(* PLC project Generated.project, CODESYS CODESYS V3.5 SP19 Patch 1 *)
(* stored: creationDateTime 2026-09-06T13:00:42.384826, modificationDateTime 2026-09-06T13:00:42.384826 *)

(* ======================================================================= 🧩 ST_Fault — Brique socle défaut (2 vues : live + latchée) ─────────────────────────────────────────────────────────────── 🎯 Rôle : porter l'état défaut d'un composant, applicable dans TOUS les cas (acquittable ou non), sans brique warning séparée. • Vue LIVE (Error / ErrorId) : suit la cause, retombe seule à 0. • Vue LATCHÉE (Latched / LatchedId): mémorisée au défaut, reste jusqu'au front Reset. Le choix acquittable / non-acquittable se fait PAR CAUSE (ST_FaultCause.Latching), jamais par bloc. 🔒 Sécurité : interlock TOUJOURS sur la cause brute (Error / ErrorId), jamais sur l'acquittement. Reset TOUJOURS effectif, jamais conditionné (std §9). 🧬 Composition : brique de base réutilisable — sortie de FB, struct métier, GVL. Texte IHM NON stocké ici : dérivé côté IHM depuis LatchedId / ErrorId. 📄 Doc : DOC/STDS/CODE_QUALITY_STANDARDS.md §2quinquies / §9 ======================================================================= *)
TYPE ST_Fault : STRUCT
  Error : BOOL;  (* <-- [DIAG] vue LIVE : au moins une cause présente maintenant *)
  ErrorId : WORD;  (* <-- [DIAG] bitfield des causes présentes maintenant (0 si aucune) *)
  Latched : BOOL;  (* <-- [DIAG] vue LATCHÉE : défaut non acquitté, reste jusqu'au front Reset *)
  LatchedId : WORD;  (* <-- [DIAG] ErrorId figé à l'apparition du défaut, effacé au Reset *)
END_STRUCT;
END_TYPE

(* ======================================================================= 🧩 ST_FaultCause — Cause élémentaire alimentant ST_Fault (socle FB_FaultCore) ─────────────────────────────────────────────────────────────── 🎯 Rôle : une cause exprimée EN CLAIR (BOOL + libellé), sans bitfield ni masque. Le FB métier remplit une liste (ARRAY[0..15] OF ST_FaultCause) ; le socle FB_FaultCore en déduit ST_Fault (vue live + vue latchée). 🔒 Sécurité : interlock TOUJOURS sur Active (cause brute), jamais sur le latch. Latching = TRUE → la cause ARME la vue latchée (défaut à acquitter). Latching = FALSE → la cause n'alimente que la vue live (retombe seule). Fail-safe : une cause laissée à Latching=FALSE reste visible en live — pour la rendre acquittable, il faut le déclarer explicitement. 📄 Doc : DOC/STDS/CODE_QUALITY_STANDARDS.md §2quinquies / §9 ======================================================================= *)
TYPE ST_FaultCause : STRUCT
  Active : BOOL;  (* 1 = cause présente maintenant (interlock sur cette valeur) *)
  Latching : BOOL;  (* 1 = cause à acquitter (arme Latched) ; 0 = live seulement *)
  Texte : STRING;  (* libellé prêt IHM (non stocké dans ST_Fault, dérivé côté IHM) *)
END_STRUCT;
END_TYPE

(* ======================================================================= 🛡️ FB_Encoder_Safety — Bornage physique & surveillance cohérence ─────────────────────────────────────────────────────────────── 🎯 Rôle : Bornage physique absolu [-99; +99]m et relais d'incohérence redémarrage 🔒 Polarité : EncoderIncoherent=TRUE en cas de hors bornes ou HomingSuspect 🛡️ Sécurité : Verrouillage de la position câble sûre 📄 Doc métier : DOC/AF/AF_Partie-09_Fonction_Encoder_v2.4.md ======================================================================= *)
FUNCTION_BLOCK FB_Encoder_Safety
  VAR_INPUT
    Enable : BOOL;  (* === COMMANDES & AUTORISATIONS === --> [CMD] Autorisation generale FB (TRUE=Autorise) *)
    Reset : BOOL;  (* --> [CMD] Acquittement defaut (front montant) *)
    CablePosM : REAL;  (* === MESURES & ALERTE HOMING === --> [HW] Position calculee (m, sortie FB_Encoder_Scale) *)
    HomingSuspect : BOOL;  (* --> [SAFE] Alerte incoherence redemarrage (FB_Encoder_Homing) *)
    PositionMinM : REAL := -99;  (* === REGLAGES & BORNES PHYSIQUES === --> [CFG] Plafond bornage physique bas (m) *)
    PositionMaxM : REAL := 99;  (* --> [CFG] Plafond bornage physique haut (m) *)
    BypassGlobal : BOOL := FALSE;  (* === TESTS & BYPASS === --> [TST] Neutralisation defaut de bornage pour mise en service *)
  END_VAR
  VAR_OUTPUT
    Ready : BOOL;  (* === ETATS IEC & SYNOPTIQUE === <-- [STAT] FB pret a fonctionner *)
    Fault : ST_Fault;  (* 🧩 Statut transverse (forme cible ST_Fault) *)
    CablePosMSafe : REAL;  (* === MESURES SURE & SECURITE === <-- [DIAG] Position cable instantanee transmise (m) *)
    EncoderIncoherent : BOOL;  (* <-- [SAFE] Incoherence ou hors bornes (TRUE = defaut) *)
  END_VAR
  VAR
    ResetEdge : R_TRIG;  (* === DETECTEURS DE FRONT === . [LOC] Detecteur front montant Reset *)
    instFault : FB_FaultCore;  (* === SOCLE DEFAUT (FB_FaultCore) === * [INST] Socle défaut transverse *)
    instCauses : ARRAY[0..15] OF ST_FaultCause;  (* . [LOC] Table des causes nommées *)
  END_VAR

            

// === IMPLEMENTATION ===

{region "§1 Causes & Socle Défaut (évalué en continu)"}
// 🔑 1. RESET FRONT
ResetEdge(CLK := Reset);

// 🔍 2. SURVEILLANCE BORNAGE & INCOHÉRENCE BOOT
instCauses[0].Active   := NOT BypassGlobal AND ((CablePosM < PositionMinM) OR (CablePosM > PositionMaxM));
instCauses[0].Latching := FALSE;
instCauses[0].Texte    := 'Depassement bornes physiques absolues cable';

instCauses[1].Active   := NOT BypassGlobal AND HomingSuspect;
instCauses[1].Latching := FALSE;
instCauses[1].Texte    := 'Incoherence position au redemarrage';

// Appel du socle de défaut
instFault(Enable := Enable, Reset := Reset, Causes := instCauses);
Fault := instFault.Fault;
{endregion}

{region "§2 Gate neutralisation"}
// 🛑 2. GATE
IF NOT Enable THEN
    Ready := FALSE;
    CablePosMSafe := CablePosM;
    EncoderIncoherent := FALSE;
    RETURN;
END_IF;

Ready := Enable AND NOT Fault.Latched;
{endregion}

{region "§3 Transmission mesure et sécurité"}
// 📏 3. TRANSMISSION DE LA MESURE & SÉCURITÉ
CablePosMSafe := CablePosM;
EncoderIncoherent := Fault.Error;
{endregion}

          
END_FUNCTION_BLOCK

(* ======================================================================= 🧩 FB_FaultCore — Socle de remplissage de ST_Fault (vue live + vue latchée) ─────────────────────────────────────────────────────────────── 🎯 Rôle : à partir d'une LISTE de causes en clair (ARRAY[0..15] OF ST_FaultCause), produire la brique ST_Fault : • Error / ErrorId : vue LIVE, suit les causes Active, retombe seule. • Latched / LatchedId: vue LATCHÉE, chaque bit figé à l'apparition d'une cause `Active AND Latching`, conservé jusqu'au front Reset. 🔒 Sécurité : - interlock TOUJOURS sur `Causes[i].Active` (cause brute), jamais sur le latch. - Reset TOUJOURS effectif, jamais conditionné (std §9) — agit même Enable=FALSE. - Latching=FALSE → cause visible en LIVE seulement (fail-safe : reste visible). - un défaut laté non acquitté reste publié même FB désactivé (pas d'effacement silencieux sur bascule Enable OFF→ON sans Reset). - une cause à acquitter réapparue re-arme son bit (ré-alarme). 🧬 Un seul socle, réutilisé par tout FB `standard` qui expose un ST_Fault. Pas de State, pas de Warning, pas de texte — hors périmètre de ce socle. 📄 Doc : DOC/STDS/CODE_QUALITY_STANDARDS.md §2quinquies / §9 ======================================================================= *)
FUNCTION_BLOCK FB_FaultCore
  VAR_INPUT
    Enable : BOOL;  (* --> [CMD] Autorisation générale du FB porteur *)
    Reset : BOOL;  (* --> [CMD] Front d'acquittement (jamais conditionné, §9) *)
    Causes : ARRAY[0..15] OF ST_FaultCause;  (* --> [CMD] Liste des causes en clair (Active / Latching / Texte) *)
  END_VAR
  VAR_OUTPUT
    Ready : BOOL;  (* <-- [STAT] FB porteur autorisé (= Enable) *)
    Fault : ST_Fault;  (* <-- [DIAG] Brique défaut (mappée 1:1 sur la sortie du FB porteur) *)
  END_VAR
  VAR
    ResetEdge : R_TRIG;  (* . [LOC] Front montant Reset *)
    Latch : ARRAY[0..15] OF BOOL;  (* . [LOC] Bit laté par cause, jusqu'au Reset *)
    i : INT;  (* . [LOC] Index de parcours de la liste *)
  END_VAR

            

{region "§1 Reset (front, toujours effectif)"}
// Front Reset : efface tous les latches. Jamais conditionné, agit même Enable=FALSE (§9).
Ready := Enable;
ResetEdge(CLK := Reset);
IF ResetEdge.Q THEN
    FOR i := 0 TO 15 DO Latch[i] := FALSE; END_FOR;
END_IF;
{endregion}

{region "§2 Vue LIVE — Error / ErrorId"}
// Bitfield des causes présentes MAINTENANT. Retombe seule à 0 quand les causes disparaissent.
// Non évaluée si Enable=FALSE (pas de lecture de cause hors autorisation).
Fault.ErrorId := 0;
IF Enable THEN
    FOR i := 0 TO 15 DO
        IF Causes[i].Active THEN
            Fault.ErrorId := Fault.ErrorId OR SHL(WORD#1, INT_TO_DWORD(i));
        END_IF;
    END_FOR;
END_IF;
Fault.Error := (Fault.ErrorId <> 0);
{endregion}

{region "§3 Armement des latches (causes à acquitter)"}
// Une cause Active ET Latching arme son bit ; le bit reste jusqu'au front Reset (§1),
// même si la cause disparaît. Réapparition => ré-armement (ré-alarme).
IF Enable THEN
    FOR i := 0 TO 15 DO
        IF Causes[i].Active AND Causes[i].Latching THEN
            Latch[i] := TRUE;
        END_IF;
    END_FOR;
END_IF;
{endregion}

{region "§4 Vue LATCHÉE — Latched / LatchedId"}
// Toujours publiée, y compris Enable=FALSE : un défaut non acquitté reste visible.
Fault.LatchedId := 0;
FOR i := 0 TO 15 DO
    IF Latch[i] THEN
        Fault.LatchedId := Fault.LatchedId OR SHL(WORD#1, INT_TO_DWORD(i));
    END_IF;
END_FOR;
Fault.Latched := (Fault.LatchedId <> 0);
{endregion}

          
END_FUNCTION_BLOCK
